PROGRAM MAIN_SFC
VAR
	Timer			: TON;
	fbSFC_SamplePOU : FB_SFC_SamplePou;

	eOperation		: E_Operation := eOp_Add;
	iResultC		: DINT;
	bZero			: BOOL;
	bPos			: BOOL;
	bNeg			: BOOL;
	bTest			: BOOL;
	tTimerValue		: TIME := T#3S;
END_VAR

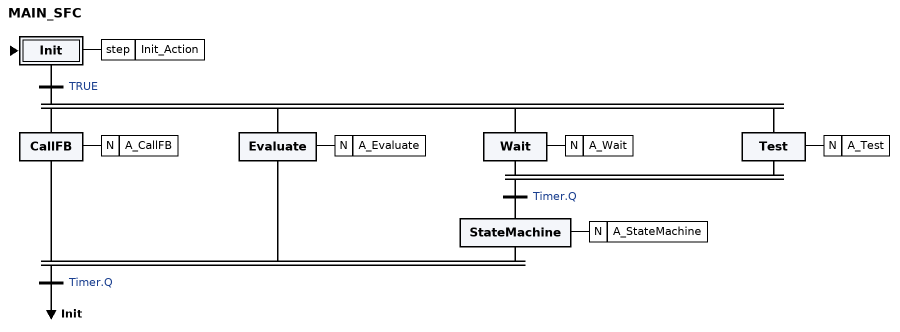
INITIAL_STEP Init:
    Init_Action(N);  // step action
END_STEP
TRANSITION FROM Init TO (CallFB, Evaluate, Wait, Test)
    := TRUE;
END_TRANSITION
STEP CallFB:
    A_CallFB(N);
END_STEP
STEP Evaluate:
    A_Evaluate(N);
END_STEP
STEP Wait:
    A_Wait(N);
END_STEP
STEP Test:
    A_Test(N);
END_STEP
TRANSITION FROM (Wait, Test) TO StateMachine
    := Timer.Q;
END_TRANSITION
STEP StateMachine:
    A_StateMachine(N);
END_STEP
TRANSITION FROM (CallFB, Evaluate, StateMachine) TO Init
    := Timer.Q;
END_TRANSITION

ACTION A_CallFB:
(* FB Call *)
fbSFC_SamplePOU(
	eOperation	:= eOperation,
	iResultC	=> iResultC
);
END_ACTION

ACTION A_Evaluate:
(* Evaluation *)
IF fbSFC_SamplePOU.iResultC = 0 THEN
	bZero := TRUE;
	bPos := FALSE;
	bNeg := FALSE;
ELSIF fbSFC_SamplePOU.iResultC > 0 THEN
	bZero := FALSE;
	bPos := TRUE;
	bNeg := FALSE;
ELSIF fbSFC_SamplePOU.iResultC < 0 THEN
	bZero := FALSE;
	bPos := FALSE;
	bNeg := TRUE;
END_IF
END_ACTION

ACTION A_StateMachine:
(* State machine *)
CASE eOperation OF
eOp_Add:
	eOperation := eOp_MUL;
eOp_Sub:
	eOperation := eOp_ADD;
eOp_Mul:
	eOperation := eOp_SUB;
END_CASE
END_ACTION

ACTION A_Test:
bTest := (((bZero AND bPos) OR (bPos XOR bNeg)) AND (Timer.ET > TIME#500MS) AND (iResultC <= 0)) OR (Timer.ET <= TIME#500MS);
END_ACTION

ACTION A_Wait:
(* Timer *)
Timer(IN := TRUE, PT := tTimerValue);
END_ACTION

ACTION Init_Action:
Timer(IN := FALSE);
END_ACTION

END_PROGRAM

(* stored: Version 1.1.0.1, ProductVersion 3.1.4024.11
   POU MAIN_SFC: Id {54c1c195-7323-4bcb-81ad-ac55cad23ac1}, SpecialFunc None
   Action A_CallFB: Id {fb1521e1-843b-4e41-852c-872d9a7cef9d}
   Action A_Evaluate: Id {54b4f0c5-01a0-48df-9726-32d51c0eced9}
   Action A_StateMachine: Id {72b5b7cd-e968-4af9-a5c2-045dc6b17163}
   Action A_Test: Id {56fab01f-8691-416c-a76b-d34c0b043b8f}
   Action A_Wait: Id {913d10b4-2bd9-4fb8-9bd0-f1345984d5f9}
   Action Init_Action: Id {1d826b43-913e-4ca2-a2ff-1162caa117cf} *)
